Yaskawa INFORM job: LOGIC_TEST.JBI

/JOB
//NAME LOGIC_TEST
//POS
///NPOS 0,0,0,0,0,0
//INST
///DATE 2021/12/03 12:01
///ATTR SC,RW
///GROUP1 RB1
NOP
CALL JOB:SYS_SPINDLE_START
WAIT T=5.00
CALL JOB:SYS_SPINDLE_STOP
END
